// SIMATIC S7-200 project (STEP 7-Micro/WIN), CPU 224XP REL 02.01

SYMBOL_TABLE USER1
start            I0.0     // khoi dong he thong
stopp            I0.1     // dung he thong
s1               I0.2     // cam bien nguoi/vat
s2               I0.3     // cam bien mo cua
s3               I0.4     // cam bien dong cua
k1               Q0.0     // mo cua
k2               Q0.1     // dong cua
END_SYMBOL_TABLE

ORGANIZATION_BLOCK MAIN:OB1
TITLE=PROGRAM COMMENTS
BEGIN
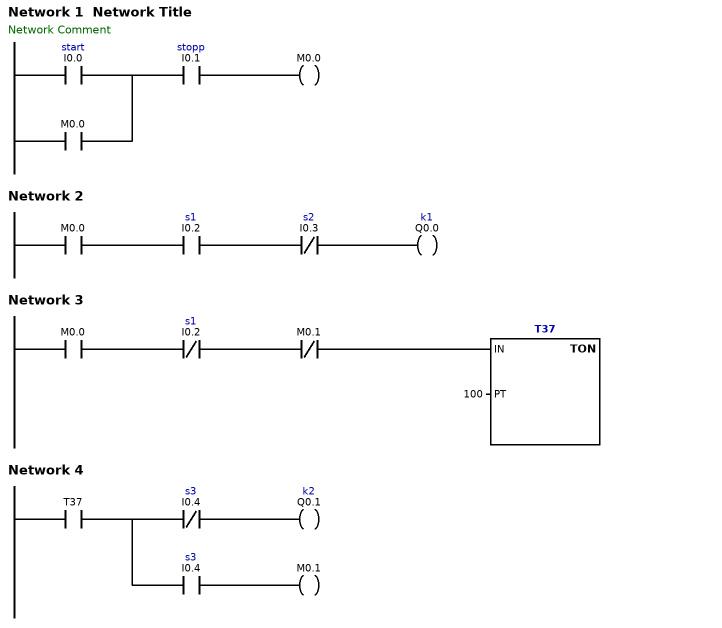
Network 1 // Network Title
// Network Comment
LD     start:I0.0
O      M0.0
A      stopp:I0.1
=      M0.0
Network 2
LD     M0.0
A      s1:I0.2
AN     s2:I0.3
=      k1:Q0.0
Network 3
LD     M0.0
AN     s1:I0.2
AN     M0.1
TON    T37, 100
Network 4
LD     T37
LPS
AN     s3:I0.4
=      k2:Q0.1
LPP
A      s3:I0.4
=      M0.1
END_ORGANIZATION_BLOCK
